# B&R Automation Studio project CombinedLinenSoiledA9KAN (part 10)

```iecst
			//###DK2012Jan12
			// Set statistic.
			IF _wPrevMsgStatisticSelect <> IFmnMsg.In.wMsgStatisticSelect THEN
				_wPrevMsgStatisticSelect := IFmnMsg.In.wMsgStatisticSelect;
				_xMsgStatisticSelectChanged := TRUE;
			END_IF;

			IF IFmnMsg.Trig.xRefreshStatistic OR _xRefreshStatistic THEN
				_msgStatisticNumShowIdx := _msgStatisticNumIdx;
				_msgStatisticTimeShowIdx := _msgStatisticTimeIdx;
				_wIFMsgStatisticCntNumShow := _wIFMsgStatisticCntNum;
				_wIFMsgStatisticCntTimeShow := _wIFMsgStatisticCntTime;
				IFmnMsg.Trig.xRefreshStatistic := FALSE;
				_xRefreshStatistic := FALSE;
				_xMsgStatisticSelectChanged := TRUE;
			END_IF;

			IF _xMsgStatisticSelectChanged THEN
				IF IFmnMsg.In.wMsgStatisticSelect = 0 THEN
					IFmnMsg.Out.wMsgStatisticCnt := _wIFMsgStatisticCntNumShow;
					FOR _wMsgListCnt := 0 TO MNMSG_MAX_IDX_VCMSGSTATLIST BY 1 DO
						_utfMsgTextTempFirst := UINT_TO_WSTRING(_msgStatisticNumShowIdx[_wMsgListCnt].wFunction_ID);
						_utfMsgTextTempSecond := ".";
						brwcsncat(ADR(_utfMsgTextTempFirst), ADR(_utfMsgTextTempSecond),
						UDINT_TO_UINT(brwcslen(ADR(_utfMsgTextTempSecond)) - (brwcslen(ADR(_utfMsgTextTempFirst)) + brwcslen(ADR(_utfMsgTextTempSecond)) - (SIZEOF(_utfMsgTextTempFirst) / 2 - 1))));
						_utfMsgTextTempSecond := UINT_TO_WSTRING(_msgStatisticNumShowIdx[_wMsgListCnt].wMsgNumber);
						brwcsncat(ADR(_utfMsgTextTempFirst), ADR(_utfMsgTextTempSecond),
						UDINT_TO_UINT(brwcslen(ADR(_utfMsgTextTempSecond)) - (brwcslen(ADR(_utfMsgTextTempFirst)) + brwcslen(ADR(_utfMsgTextTempSecond)) - (SIZEOF(_utfMsgTextTempFirst) / 2 - 1))));
						_utfMsgTextTempSecond := ".";
						brwcsncat(ADR(_utfMsgTextTempFirst), ADR(_utfMsgTextTempSecond),
						UDINT_TO_UINT(brwcslen(ADR(_utfMsgTextTempSecond)) - (brwcslen(ADR(_utfMsgTextTempFirst)) + brwcslen(ADR(_utfMsgTextTempSecond)) - (SIZEOF(_utfMsgTextTempFirst) / 2 - 1))));
						_utfMsgTextTempSecond := UINT_TO_WSTRING(_msgStatisticNumShowIdx[_wMsgListCnt].wInstance);
						brwcsncat(ADR(_utfMsgTextTempFirst), ADR(_utfMsgTextTempSecond),
						UDINT_TO_UINT(brwcslen(ADR(_utfMsgTextTempSecond)) - (brwcslen(ADR(_utfMsgTextTempFirst)) + brwcslen(ADR(_utfMsgTextTempSecond)) - (SIZEOF(_utfMsgTextTempFirst) / 2 - 1))));
						_utfMsgTextTempSecond := " ";
						brwcsncat(ADR(_utfMsgTextTempFirst), ADR(_utfMsgTextTempSecond),
						UDINT_TO_UINT(brwcslen(ADR(_utfMsgTextTempSecond)) - (brwcslen(ADR(_utfMsgTextTempFirst)) + brwcslen(ADR(_utfMsgTextTempSecond)) - (SIZEOF(_utfMsgTextTempFirst) / 2 - 1))));
						_wActFunctionID := _msgStatisticNumShowIdx[_wMsgListCnt].wFunction_ID;
						_wActMsgNumber := _msgStatisticNumShowIdx[_wMsgListCnt].wMsgNumber;
						_wActInstance := _msgStatisticNumShowIdx[_wMsgListCnt].wInstance;
						_actGetTxtFim;
						IF NOT((_wActFunctionID = 0) OR (_wActMsgNumber = 0)) THEN
							IFmnMsg.Out.MsgStatistic[_wMsgListCnt].utfMsgText := _utfMsgTextTempFirst;
							IFmnMsg.Out.MsgStatistic[_wMsgListCnt].lValue := _msgStatisticNumShowIdx[_wMsgListCnt].lValue;
						ELSE
							IFmnMsg.Out.MsgStatistic[_wMsgListCnt].utfMsgText := "";
							IFmnMsg.Out.MsgStatistic[_wMsgListCnt].lValue := 0;
						END_IF;
					END_FOR;
				END_IF;
				IF IFmnMsg.In.wMsgStatisticSelect = 1 THEN
					IFmnMsg.Out.wMsgStatisticCnt := _wIFMsgStatisticCntTimeShow;
					FOR _wMsgListCnt := 0 TO MNMSG_MAX_IDX_VCMSGSTATLIST BY 1 DO
						_utfMsgTextTempFirst := UINT_TO_WSTRING(_msgStatisticTimeShowIdx[_wMsgListCnt].wFunction_ID);
						_utfMsgTextTempSecond := ".";
						brwcsncat(ADR(_utfMsgTextTempFirst), ADR(_utfMsgTextTempSecond),
						UDINT_TO_UINT(brwcslen(ADR(_utfMsgTextTempSecond)) - (brwcslen(ADR(_utfMsgTextTempFirst)) + brwcslen(ADR(_utfMsgTextTempSecond)) - (SIZEOF(_utfMsgTextTempFirst) / 2 - 1))));
						_utfMsgTextTempSecond := UINT_TO_WSTRING(_msgStatisticTimeShowIdx[_wMsgListCnt].wMsgNumber);
						brwcsncat(ADR(_utfMsgTextTempFirst), ADR(_utfMsgTextTempSecond),
						UDINT_TO_UINT(brwcslen(ADR(_utfMsgTextTempSecond)) - (brwcslen(ADR(_utfMsgTextTempFirst)) + brwcslen(ADR(_utfMsgTextTempSecond)) - (SIZEOF(_utfMsgTextTempFirst) / 2 - 1))));
						_utfMsgTextTempSecond := ".";
						brwcsncat(ADR(_utfMsgTextTempFirst), ADR(_utfMsgTextTempSecond),
						UDINT_TO_UINT(brwcslen(ADR(_utfMsgTextTempSecond)) - (brwcslen(ADR(_utfMsgTextTempFirst)) + brwcslen(ADR(_utfMsgTextTempSecond)) - (SIZEOF(_utfMsgTextTempFirst) / 2 - 1))));
						_utfMsgTextTempSecond := UINT_TO_WSTRING(_msgStatisticTimeShowIdx[_wMsgListCnt].wInstance);
						brwcsncat(ADR(_utfMsgTextTempFirst), ADR(_utfMsgTextTempSecond),
						UDINT_TO_UINT(brwcslen(ADR(_utfMsgTextTempSecond)) - (brwcslen(ADR(_utfMsgTextTempFirst)) + brwcslen(ADR(_utfMsgTextTempSecond)) - (SIZEOF(_utfMsgTextTempFirst) / 2 - 1))));
						_utfMsgTextTempSecond := " ";
						brwcsncat(ADR(_utfMsgTextTempFirst), ADR(_utfMsgTextTempSecond),
						UDINT_TO_UINT(brwcslen(ADR(_utfMsgTextTempSecond)) - (brwcslen(ADR(_utfMsgTextTempFirst)) + brwcslen(ADR(_utfMsgTextTempSecond)) - (SIZEOF(_utfMsgTextTempFirst) / 2 - 1))));
						_wActFunctionID := _msgStatisticTimeShowIdx[_wMsgListCnt].wFunction_ID;
						_wActMsgNumber := _msgStatisticTimeShowIdx[_wMsgListCnt].wMsgNumber;
						_wActInstance := _msgStatisticTimeShowIdx[_wMsgListCnt].wInstance;
						_actGetTxtFim;
						IF NOT ((_wActFunctionID = 0) OR (_wActMsgNumber = 0)) THEN
							IFmnMsg.Out.MsgStatistic[_wMsgListCnt].utfMsgText := _utfMsgTextTempFirst;
							IFmnMsg.Out.MsgStatistic[_wMsgListCnt].lValue := _msgStatisticTimeShowIdx[_wMsgListCnt].lValue;
						ELSE
							IFmnMsg.Out.MsgStatistic[_wMsgListCnt].utfMsgText := "";
							IFmnMsg.Out.MsgStatistic[_wMsgListCnt].lValue := 0;
						END_IF;
					END_FOR;
				END_IF;
				_xMsgStatisticSelectChanged := FALSE;
			END_IF;
			//###DK2012Jan12

		END_IF

	ELSE	// _Plausibility.xOK

		// Horning for 500ms. After it has finished it will start again ten seconds later.
		_tonCrit1(IN := NOT _tonCrit2.Q, PT := T#500ms);
		_tonCrit2(IN := _tonCrit1.Q, PT := T#10s);

		IFmnMsg.Out.bHorn := SEL(NOT _tonCrit1.Q, 0, 1);	// Causes some horning now.

		IFmnMsg.Out.bLight := 1;

		// Meldung setzen

		IF _xNotOkFirstScan THEN

			_xNotOkFirstScan := FALSE;

			// Meldungsliste füllen

			brsmemset (ADR(mnMsgStatAd.Msg), 0, SIZEOF (mnMsgStatAd.Msg));

			_InsertMsgLine.AdrIntFaultList := ADR(mnMsgStatAd.Msg.MsgListFaultInt);
			_InsertMsgLine.AdrCntIntFault := ADR(mnMsgStatAd.Msg.MsgCntFaultInt);

			_dtHelp(enable := TRUE);

			_InsertMsgLine.Class := MNMSG_CLASS_INTFAULT;
			_InsertMsgLine.Insert := TRUE;
			_InsertMsgLine.MsgLine.bAckLevel := MNMSG_CLASS_NO_ACK;
			_InsertMsgLine.MsgLine.bInstance := 0;
			_InsertMsgLine.MsgLine.diAttr1 := 0;
			_InsertMsgLine.MsgLine.wFunction_ID := 2;
			_InsertMsgLine.MsgLine.wMsgNumber := MNMSG_MSG_SYSTEMFAULT;
			_InsertMsgLine.MsgLine.TimeStamp := _dtHelp.DT1;
			_InsertMsgLine();

			mnMsgStatAd.Msg.dtMsgIntFaultChanged := _dtHelp.DT1;

		END_IF

	END_IF;	// IFmnMsg.Out.xMnMsgReady

	////////////////////////////////////////////////////////////////////////////////////////////////////////////////////////////////////////////////////////////////////////////////////////////////////////////////////////////////////////////////////////////////////////////////////////////////////////////////////////////////////////////////////////////////////////////////////////////////////////////////////////////////////////////////////////////////////////////////////////////////////////////////////////////////////////////////////////////////////////////////////////////////////////////////////////////////////

	_LastExecute(enable := TRUE);
	_dtLastExecute := _LastExecute.DT1;

END_PROGRAM
```

#### _actGetTxtFim.st
```iecst
(********************************************************************
 * COPYRIGHT -- Herbert Kannegiesser GmbH
 ********************************************************************
 * Program: mnMsg
 * File: actGetTxtFim.st
 * Author: kuehne
 * Created: February 21, 2012
 ********************************************************************
 * Implementation of program mnMsg
 ********************************************************************)

(* Add a new action to your IEC program or library *)
ACTION _actGetTxtFim:
	IF _xMnTxtReady THEN
		_MsgTxtLine ACCESS IFmnTxt.Out.ptrFunctionTxtList;
		_BinSearchTxt.MsgTxtList := IFmnTxt.Out.ptrFunctionTxtList;
		_BinSearchTxt.wCntMsgTxt := IFmnTxt.Out.wCntFunctionTxt;
		_BinSearchTxt.wFunctionID := _wActFunctionID;
		_BinSearchTxt.wNumber := _wActMsgNumber;
		_BinSearchTxt.wInstance := _wActInstance;
		_BinSearchTxt.bTupel := 1;
		_BinSearchTxt();
		IF _BinSearchTxt.wStatus <> ERR_OK THEN
			brwcscat(ADR(_utfMsgTextTempFirst), ADR(""));
		ELSE
			_wTxtIdx := _BinSearchTxt.wMsgPos;
			_BinSearchCfg.wFunctionID := _wActFunctionID;
			_BinSearchCfg.wMsgNo := _wActMsgNumber;
			_BinSearchCfg.wInstance := _wActInstance;
			_BinSearchCfg();
			IF _BinSearchCfg.wStatus = ERR_OK THEN
				_wImageIdx := _BinSearchCfg.wMsgIdx;
				_utfMsgTextTempThird := "";
				_utfMsgTextTempThird := DINT_TO_WSTRING(_MsgImage[_wImageIdx].diMsgAttr1);
			ELSE
				_utfMsgTextTempThird := "{##AttrVar1}";
			END_IF;
			_utfMsgTextTempSecond := "";
			_fbMsgReplSubStr.utfStr := ADR(_MsgTxtLine[_wTxtIdx].utfText);
			_fbMsgReplSubStr.utfSubStr := ADR("{##AttrVar1}");
			_fbMsgReplSubStr.utfStrToReplWith := ADR(_utfMsgTextTempThird);
			_fbMsgReplSubStr.utfStrResult := ADR(_utfMsgTextTempSecond);
			_fbMsgReplSubStr();
			IF _BinSearchCfg.wStatus = ERR_OK THEN
				_wImageIdx := _BinSearchCfg.wMsgIdx;
				_utfMsgTextTempThird := "";
				_utfMsgTextTempThird := DINT_TO_WSTRING(_MsgImage[_wImageIdx].diMsgAttr2);
			ELSE
				_utfMsgTextTempThird := "{##AttrVar2}";
			END_IF;
			_utfMsgTextTempFourth := "";
			_utfMsgTextTempFourth := _utfMsgTextTempSecond;
			_utfMsgTextTempSecond := "";
			_fbMsgReplSubStr.utfStr := ADR(_utfMsgTextTempFourth);
			_fbMsgReplSubStr.utfSubStr := ADR("{##AttrVar2}");
			_fbMsgReplSubStr.utfStrToReplWith := ADR(_utfMsgTextTempThird);
			_fbMsgReplSubStr.utfStrResult := ADR(_utfMsgTextTempSecond);
			_fbMsgReplSubStr();
			IF _BinSearchCfg.wStatus = ERR_OK THEN
				_wImageIdx := _BinSearchCfg.wMsgIdx;
				_utfMsgTextTempThird := "";
				_utfMsgTextTempThird := STRING_TO_WSTRING(_MsgImage[_wImageIdx].sMsgAttrTxt);
			ELSE
				_utfMsgTextTempThird := "{##AttrTxt}";
			END_IF;
			_utfMsgTextTempFourth := "";
			_utfMsgTextTempFourth := _utfMsgTextTempSecond;
			_utfMsgTextTempSecond := "";
			_fbMsgReplSubStr.utfStr := ADR(_utfMsgTextTempFourth);
			_fbMsgReplSubStr.utfSubStr := ADR("{##AttrTxt}");
			_fbMsgReplSubStr.utfStrToReplWith := ADR(_utfMsgTextTempThird);
			_fbMsgReplSubStr.utfStrResult := ADR(_utfMsgTextTempSecond);
			_fbMsgReplSubStr();
			brwcsncat(ADR(_utfMsgTextTempFirst), ADR(_utfMsgTextTempSecond),
			UDINT_TO_UINT(brwcslen(ADR(_utfMsgTextTempSecond)) - (brwcslen(ADR(_utfMsgTextTempFirst)) + brwcslen(ADR(_utfMsgTextTempSecond)) - (SIZEOF(_utfMsgTextTempFirst) / 2 - 1))));
			_utfMsgTextTempSecond := "";
			_utfMsgTextTempSecond := " ";
			brwcsncat(ADR(_utfMsgTextTempFirst), ADR(_utfMsgTextTempSecond),
			UDINT_TO_UINT(brwcslen(ADR(_utfMsgTextTempSecond)) - (brwcslen(ADR(_utfMsgTextTempFirst)) + brwcslen(ADR(_utfMsgTextTempSecond)) - (SIZEOF(_utfMsgTextTempFirst) / 2 - 1))));
		END_IF;
		_MsgTxtLine ACCESS IFmnTxt.Out.ptrInstanceTxtList;
		_BinSearchTxt.MsgTxtList := IFmnTxt.Out.ptrInstanceTxtList;
		_BinSearchTxt.wCntMsgTxt := IFmnTxt.Out.wCntInstanceTxt;
		_BinSearchTxt.wFunctionID := _wActFunctionID;
		_BinSearchTxt.wNumber := _wActInstance;
		_BinSearchTxt.wInstance := 0;
		_BinSearchTxt.bTupel := 2;
		_BinSearchTxt();
		IF _BinSearchTxt.wStatus <> ERR_OK THEN
			brwcscat(ADR(_utfMsgTextTempFirst), ADR(""));
		ELSE
			_wTxtIdx := _BinSearchTxt.wMsgPos;
			_BinSearchCfg.wFunctionID := _wActFunctionID;
			_BinSearchCfg.wMsgNo := _wActMsgNumber;
			_BinSearchCfg.wInstance := _wActInstance;
			_BinSearchCfg();
			IF _BinSearchCfg.wStatus = ERR_OK THEN
				_wImageIdx := _BinSearchCfg.wMsgIdx;
				_utfMsgTextTempThird := "";
				_utfMsgTextTempThird := DINT_TO_WSTRING(_MsgImage[_wImageIdx].diMsgAttr1);
			ELSE
				_utfMsgTextTempThird := "{##AttrVar1}";
			END_IF;
			_utfMsgTextTempSecond := "";
			_fbMsgReplSubStr.utfStr := ADR(_MsgTxtLine[_wTxtIdx].utfText);
			_fbMsgReplSubStr.utfSubStr := ADR("{##AttrVar1}");
			_fbMsgReplSubStr.utfStrToReplWith := ADR(_utfMsgTextTempThird);
			_fbMsgReplSubStr.utfStrResult := ADR(_utfMsgTextTempSecond);
			_fbMsgReplSubStr();
			IF _BinSearchCfg.wStatus = ERR_OK THEN
				_wImageIdx := _BinSearchCfg.wMsgIdx;
				_utfMsgTextTempThird := "";
				_utfMsgTextTempThird := DINT_TO_WSTRING(_MsgImage[_wImageIdx].diMsgAttr2);
			ELSE
				_utfMsgTextTempThird := "{##AttrVar2}";
			END_IF;
			_utfMsgTextTempFourth := "";
			_utfMsgTextTempFourth := _utfMsgTextTempSecond;
			_utfMsgTextTempSecond := "";
			_fbMsgReplSubStr.utfStr := ADR(_utfMsgTextTempFourth);
			_fbMsgReplSubStr.utfSubStr := ADR("{##AttrVar2}");
			_fbMsgReplSubStr.utfStrToReplWith := ADR(_utfMsgTextTempThird);
			_fbMsgReplSubStr.utfStrResult := ADR(_utfMsgTextTempSecond);
			_fbMsgReplSubStr();
			IF _BinSearchCfg.wStatus = ERR_OK THEN
				_wImageIdx := _BinSearchCfg.wMsgIdx;
				_utfMsgTextTempThird := "";
				_utfMsgTextTempThird := STRING_TO_WSTRING(_MsgImage[_wImageIdx].sMsgAttrTxt);
			ELSE
				_utfMsgTextTempThird := "{##AttrTxt}";
			END_IF;
			_utfMsgTextTempFourth := "";
			_utfMsgTextTempFourth := _utfMsgTextTempSecond;
			_utfMsgTextTempSecond := "";
			_fbMsgReplSubStr.utfStr := ADR(_utfMsgTextTempFourth);
			_fbMsgReplSubStr.utfSubStr := ADR("{##AttrTxt}");
			_fbMsgReplSubStr.utfStrToReplWith := ADR(_utfMsgTextTempThird);
			_fbMsgReplSubStr.utfStrResult := ADR(_utfMsgTextTempSecond);
			_fbMsgReplSubStr();
			brwcsncat(ADR(_utfMsgTextTempFirst), ADR(_utfMsgTextTempSecond),
			UDINT_TO_UINT(brwcslen(ADR(_utfMsgTextTempSecond)) - (brwcslen(ADR(_utfMsgTextTempFirst)) + brwcslen(ADR(_utfMsgTextTempSecond)) - (SIZEOF(_utfMsgTextTempFirst) / 2 - 1))));
			_utfMsgTextTempSecond := "";
			_utfMsgTextTempSecond := " ";
			brwcsncat(ADR(_utfMsgTextTempFirst), ADR(_utfMsgTextTempSecond),
			UDINT_TO_UINT(brwcslen(ADR(_utfMsgTextTempSecond)) - (brwcslen(ADR(_utfMsgTextTempFirst)) + brwcslen(ADR(_utfMsgTextTempSecond)) - (SIZEOF(_utfMsgTextTempFirst) / 2 - 1))));
		END_IF;
		_MsgTxtLine ACCESS IFmnTxt.Out.ptrMessageTxtList;
		_BinSearchTxt.MsgTxtList := IFmnTxt.Out.ptrMessageTxtList;
		_BinSearchTxt.wCntMsgTxt := IFmnTxt.Out.wCntMessageTxt;
		_BinSearchTxt.wFunctionID := _wActFunctionID;
		_BinSearchTxt.wNumber := _wActMsgNumber;
		_BinSearchTxt.wInstance := _wActInstance;
		_BinSearchTxt.bTupel := 2;
		_BinSearchTxt();
		IF _BinSearchTxt.wStatus <> ERR_OK THEN
			brwcscat(ADR(_utfMsgTextTempFirst), ADR(""));
		ELSE
			_wTxtIdx := _BinSearchTxt.wMsgPos;
			_BinSearchCfg.wFunctionID := _wActFunctionID;
			_BinSearchCfg.wMsgNo := _wActMsgNumber;
			_BinSearchCfg.wInstance := _wActInstance;
			_BinSearchCfg();
			IF _BinSearchCfg.wStatus = ERR_OK THEN
				_wImageIdx := _BinSearchCfg.wMsgIdx;
				_utfMsgTextTempThird := "";
				_utfMsgTextTempThird := DINT_TO_WSTRING(_MsgImage[_wImageIdx].diMsgAttr1);
			ELSE
				_utfMsgTextTempThird := "{##AttrVar1}";
			END_IF;
			_utfMsgTextTempSecond := "";
			_fbMsgReplSubStr.utfStr := ADR(_MsgTxtLine[_wTxtIdx].utfText);
			_fbMsgReplSubStr.utfSubStr := ADR("{##AttrVar1}");
			_fbMsgReplSubStr.utfStrToReplWith := ADR(_utfMsgTextTempThird);
			_fbMsgReplSubStr.utfStrResult := ADR(_utfMsgTextTempSecond);
			_fbMsgReplSubStr();
			IF _BinSearchCfg.wStatus = ERR_OK THEN
				_wImageIdx := _BinSearchCfg.wMsgIdx;
				_utfMsgTextTempThird := "";
				_utfMsgTextTempThird := DINT_TO_WSTRING(_MsgImage[_wImageIdx].diMsgAttr2);
			ELSE
				_utfMsgTextTempThird := "{##AttrVar2}";
			END_IF;
			_utfMsgTextTempFourth := "";
			_utfMsgTextTempFourth := _utfMsgTextTempSecond;
			_utfMsgTextTempSecond := "";
			_fbMsgReplSubStr.utfStr := ADR(_utfMsgTextTempFourth);
			_fbMsgReplSubStr.utfSubStr := ADR("{##AttrVar2}");
			_fbMsgReplSubStr.utfStrToReplWith := ADR(_utfMsgTextTempThird);
			_fbMsgReplSubStr.utfStrResult := ADR(_utfMsgTextTempSecond);
			_fbMsgReplSubStr();
			IF _BinSearchCfg.wStatus = ERR_OK THEN
				_wImageIdx := _BinSearchCfg.wMsgIdx;
				_utfMsgTextTempThird := "";
				_utfMsgTextTempThird := STRING_TO_WSTRING(_MsgImage[_wImageIdx].sMsgAttrTxt);
			ELSE
				_utfMsgTextTempThird := "{##AttrTxt}";
			END_IF;
			_utfMsgTextTempFourth := "";
			_utfMsgTextTempFourth := _utfMsgTextTempSecond;
			_utfMsgTextTempSecond := "";
			_fbMsgReplSubStr.utfStr := ADR(_utfMsgTextTempFourth);
			_fbMsgReplSubStr.utfSubStr := ADR("{##AttrTxt}");
			_fbMsgReplSubStr.utfStrToReplWith := ADR(_utfMsgTextTempThird);
			_fbMsgReplSubStr.utfStrResult := ADR(_utfMsgTextTempSecond);
			_fbMsgReplSubStr();
			brwcsncat(ADR(_utfMsgTextTempFirst), ADR(_utfMsgTextTempSecond),
			UDINT_TO_UINT(brwcslen(ADR(_utfMsgTextTempSecond)) - (brwcslen(ADR(_utfMsgTextTempFirst)) + brwcslen(ADR(_utfMsgTextTempSecond)) - (SIZEOF(_utfMsgTextTempFirst) / 2 - 1))));
		END_IF;
	ELSE
		brwcscat(ADR(_utfMsgTextTempFirst), ADR(""));
	END_IF;
END_ACTION
```

#### _actGetTxtFimh.st
```iecst
(********************************************************************
 * COPYRIGHT -- Herbert Kannegiesser GmbH
 ********************************************************************
 * Program: mnMsg
 * File: actGetTxtFimh.st
 * Author: kuehne
 * Created: February 22, 2012
 ********************************************************************
 * Implementation of program mnMsg
 ********************************************************************)

 (* Add a new action to your IEC program or library *)
ACTION _actGetTxtFimh:
	IF _xMnTxtReady THEN
		_MsgTxtLine ACCESS IFmnTxt.Out.ptrFunctionTxtList;
		_BinSearchTxt.MsgTxtList := IFmnTxt.Out.ptrFunctionTxtList;
		_BinSearchTxt.wCntMsgTxt := IFmnTxt.Out.wCntFunctionTxt;
		_BinSearchTxt.wFunctionID := _wActFunctionID;
		_BinSearchTxt.wNumber := _wActMsgNumber;
		_BinSearchTxt.wInstance := _wActInstance;
		_BinSearchTxt.bTupel := 1;
		_BinSearchTxt();
		IF _BinSearchTxt.wStatus <> ERR_OK THEN
			brwcscat(ADR(_utfMsgTextTempFirst), ADR(""));
		ELSE
			_wTxtIdx := _BinSearchTxt.wMsgPos;
			_utfMsgTextTempSecond := "";
			_utfMsgTextTempThird := "";
			_utfMsgTextTempThird := DINT_TO_WSTRING(_diActAttr1);
			_fbMsgReplSubStr.utfStr := ADR(_MsgTxtLine[_wTxtIdx].utfText);
			_fbMsgReplSubStr.utfSubStr := ADR("{##AttrVar1}");
			_fbMsgReplSubStr.utfStrToReplWith := ADR(_utfMsgTextTempThird);
			_fbMsgReplSubStr.utfStrResult := ADR(_utfMsgTextTempSecond);
			_fbMsgReplSubStr();
			_utfMsgTextTempThird := "";
			_utfMsgTextTempFourth := "";
			_utfMsgTextTempFourth := _utfMsgTextTempSecond;
			_utfMsgTextTempSecond := "";
			_utfMsgTextTempThird := DINT_TO_WSTRING(_diActAttr2);
			_fbMsgReplSubStr.utfStr := ADR(_utfMsgTextTempFourth);
			_fbMsgReplSubStr.utfSubStr := ADR("{##AttrVar2}");
			_fbMsgReplSubStr.utfStrToReplWith := ADR(_utfMsgTextTempThird);
			_fbMsgReplSubStr.utfStrResult := ADR(_utfMsgTextTempSecond);
			_fbMsgReplSubStr();
			_utfMsgTextTempThird := "";
			_utfMsgTextTempFourth := "";
			_utfMsgTextTempFourth := _utfMsgTextTempSecond;
			_utfMsgTextTempSecond := "";
			_utfMsgTextTempThird := STRING_TO_WSTRING(_sActAttrTxt);
			_fbMsgReplSubStr.utfStr := ADR(_utfMsgTextTempFourth);
			_fbMsgReplSubStr.utfSubStr := ADR("{##AttrTxt}");
			_fbMsgReplSubStr.utfStrToReplWith := ADR(_utfMsgTextTempThird);
			_fbMsgReplSubStr.utfStrResult := ADR(_utfMsgTextTempSecond);
			_fbMsgReplSubStr();
			brwcsncat(ADR(_utfMsgTextTempFirst), ADR(_utfMsgTextTempSecond),
			UDINT_TO_UINT(brwcslen(ADR(_utfMsgTextTempSecond)) - (brwcslen(ADR(_utfMsgTextTempFirst)) + brwcslen(ADR(_utfMsgTextTempSecond)) - (SIZEOF(_utfMsgTextTempFirst) / 2 - 1))));
			_utfMsgTextTempSecond := "";
			_utfMsgTextTempSecond := " ";
			brwcsncat(ADR(_utfMsgTextTempFirst), ADR(_utfMsgTextTempSecond),
			UDINT_TO_UINT(brwcslen(ADR(_utfMsgTextTempSecond)) - (brwcslen(ADR(_utfMsgTextTempFirst)) + brwcslen(ADR(_utfMsgTextTempSecond)) - (SIZEOF(_utfMsgTextTempFirst) / 2 - 1))));
		END_IF;
		_MsgTxtLine ACCESS IFmnTxt.Out.ptrInstanceTxtList;
		_BinSearchTxt.MsgTxtList := IFmnTxt.Out.ptrInstanceTxtList;
		_BinSearchTxt.wCntMsgTxt := IFmnTxt.Out.wCntInstanceTxt;
		_BinSearchTxt.wFunctionID := _wActFunctionID;
		_BinSearchTxt.wNumber := _wActInstance;
		_BinSearchTxt.wInstance := 0;
		_BinSearchTxt.bTupel := 2;
		_BinSearchTxt();
		IF _BinSearchTxt.wStatus <> ERR_OK THEN
			brwcscat(ADR(_utfMsgTextTempFirst), ADR(""));
		ELSE
			_wTxtIdx := _BinSearchTxt.wMsgPos;
			_utfMsgTextTempSecond := "";
			_utfMsgTextTempThird := "";
			_utfMsgTextTempThird := DINT_TO_WSTRING(_diActAttr1);
			_fbMsgReplSubStr.utfStr := ADR(_MsgTxtLine[_wTxtIdx].utfText);
			_fbMsgReplSubStr.utfSubStr := ADR("{##AttrVar1}");
			_fbMsgReplSubStr.utfStrToReplWith := ADR(_utfMsgTextTempThird);
			_fbMsgReplSubStr.utfStrResult := ADR(_utfMsgTextTempSecond);
			_fbMsgReplSubStr();
			_utfMsgTextTempThird := "";
			_utfMsgTextTempFourth := "";
			_utfMsgTextTempFourth := _utfMsgTextTempSecond;
			_utfMsgTextTempSecond := "";
			_utfMsgTextTempThird := DINT_TO_WSTRING(_diActAttr2);
			_fbMsgReplSubStr.utfStr := ADR(_utfMsgTextTempFourth);
			_fbMsgReplSubStr.utfSubStr := ADR("{##AttrVar2}");
			_fbMsgReplSubStr.utfStrToReplWith := ADR(_utfMsgTextTempThird);
			_fbMsgReplSubStr.utfStrResult := ADR(_utfMsgTextTempSecond);
			_fbMsgReplSubStr();
			_utfMsgTextTempThird := "";
			_utfMsgTextTempFourth := "";
			_utfMsgTextTempFourth := _utfMsgTextTempSecond;
			_utfMsgTextTempSecond := "";
			_utfMsgTextTempThird := STRING_TO_WSTRING(_sActAttrTxt);
			_fbMsgReplSubStr.utfStr := ADR(_utfMsgTextTempFourth);
			_fbMsgReplSubStr.utfSubStr := ADR("{##AttrTxt}");
			_fbMsgReplSubStr.utfStrToReplWith := ADR(_utfMsgTextTempThird);
			_fbMsgReplSubStr.utfStrResult := ADR(_utfMsgTextTempSecond);
			_fbMsgReplSubStr();
			brwcsncat(ADR(_utfMsgTextTempFirst), ADR(_utfMsgTextTempSecond),
			UDINT_TO_UINT(brwcslen(ADR(_utfMsgTextTempSecond)) - (brwcslen(ADR(_utfMsgTextTempFirst)) + brwcslen(ADR(_utfMsgTextTempSecond)) - (SIZEOF(_utfMsgTextTempFirst) / 2 - 1))));
			_utfMsgTextTempSecond := "";
			_utfMsgTextTempSecond := " ";
			brwcsncat(ADR(_utfMsgTextTempFirst), ADR(_utfMsgTextTempSecond),
			UDINT_TO_UINT(brwcslen(ADR(_utfMsgTextTempSecond)) - (brwcslen(ADR(_utfMsgTextTempFirst)) + brwcslen(ADR(_utfMsgTextTempSecond)) - (SIZEOF(_utfMsgTextTempFirst) / 2 - 1))));
		END_IF;
		_MsgTxtLine ACCESS IFmnTxt.Out.ptrMessageTxtList;
		_BinSearchTxt.MsgTxtList := IFmnTxt.Out.ptrMessageTxtList;
		_BinSearchTxt.wCntMsgTxt := IFmnTxt.Out.wCntMessageTxt;
		_BinSearchTxt.wFunctionID := _wActFunctionID;
		_BinSearchTxt.wNumber := _wActMsgNumber;
		_BinSearchTxt.wInstance := _wActInstance;
		_BinSearchTxt.bTupel := 2;
		_BinSearchTxt();
		IF _BinSearchTxt.wStatus <> ERR_OK THEN
			brwcscat(ADR(_utfMsgTextTempFirst), ADR(""));
		ELSE
			_wTxtIdx := _BinSearchTxt.wMsgPos;
			_utfMsgTextTempSecond := "";
			_utfMsgTextTempThird := "";
			_utfMsgTextTempThird := DINT_TO_WSTRING(_diActAttr1);
			_fbMsgReplSubStr.utfStr := ADR(_MsgTxtLine[_wTxtIdx].utfText);
			_fbMsgReplSubStr.utfSubStr := ADR("{##AttrVar1}");
			_fbMsgReplSubStr.utfStrToReplWith := ADR(_utfMsgTextTempThird);
			_fbMsgReplSubStr.utfStrResult := ADR(_utfMsgTextTempSecond);
			_fbMsgReplSubStr();
			_utfMsgTextTempThird := "";
			_utfMsgTextTempFourth := "";
			_utfMsgTextTempFourth := _utfMsgTextTempSecond;
			_utfMsgTextTempSecond := "";
			_utfMsgTextTempThird := DINT_TO_WSTRING(_diActAttr2);
			_fbMsgReplSubStr.utfStr := ADR(_utfMsgTextTempFourth);
			_fbMsgReplSubStr.utfSubStr := ADR("{##AttrVar2}");
			_fbMsgReplSubStr.utfStrToReplWith := ADR(_utfMsgTextTempThird);
			_fbMsgReplSubStr.utfStrResult := ADR(_utfMsgTextTempSecond);
			_fbMsgReplSubStr();
			_utfMsgTextTempThird := "";
			_utfMsgTextTempFourth := "";
			_utfMsgTextTempFourth := _utfMsgTextTempSecond;
			_utfMsgTextTempSecond := "";
			_utfMsgTextTempThird := STRING_TO_WSTRING(_sActAttrTxt);
			_fbMsgReplSubStr.utfStr := ADR(_utfMsgTextTempFourth);
			_fbMsgReplSubStr.utfSubStr := ADR("{##AttrTxt}");
			_fbMsgReplSubStr.utfStrToReplWith := ADR(_utfMsgTextTempThird);
			_fbMsgReplSubStr.utfStrResult := ADR(_utfMsgTextTempSecond);
			_fbMsgReplSubStr();
			brwcsncat(ADR(_utfMsgTextTempFirst), ADR(_utfMsgTextTempSecond),
			UDINT_TO_UINT(brwcslen(ADR(_utfMsgTextTempSecond)) - (brwcslen(ADR(_utfMsgTextTempFirst)) + brwcslen(ADR(_utfMsgTextTempSecond)) - (SIZEOF(_utfMsgTextTempFirst) / 2 - 1))));
		END_IF;
		// wcscat(ADR(_utfMsgTextTempFirst), ADR("internal error"));	//Also for test
		_MsgHelpTxtLine ACCESS IFmnTxt.Out.ptrMessageHelpTxtList;
		_BinSearchHelpTxt.MsgHelpTxtList := IFmnTxt.Out.ptrMessageHelpTxtList;
		_BinSearchHelpTxt.wCntMsgHelpTxt := IFmnTxt.Out.wCntMessageHlpTxt;
		_BinSearchHelpTxt.wFunctionID := _wActFunctionID;
		_BinSearchHelpTxt.wNumber := _wActMsgNumber;
		_BinSearchHelpTxt.wInstance := _wActInstance;
		_BinSearchHelpTxt.bTupel := 2;
		_BinSearchHelpTxt();
		IF _BinSearchHelpTxt.wStatus <> ERR_OK THEN
			_utfMsgTextTempSecond := "";
		ELSE
			_wTxtIdx := _BinSearchHelpTxt.wMsgPos;
			_utfMsgTextTempSecond := "";
			_utfMsgTextTempThird := "";
			_utfMsgTextTempThird := DINT_TO_WSTRING(_diActAttr1);
			_fbMsgReplSubStr.utfStr := ADR(_MsgHelpTxtLine[_wTxtIdx].utfText);
			_fbMsgReplSubStr.utfSubStr := ADR("{##AttrVar1}");
			_fbMsgReplSubStr.utfStrToReplWith := ADR(_utfMsgTextTempThird);
			_fbMsgReplSubStr.utfStrResult := ADR(_utfMsgTextTempSecond);
			_fbMsgReplSubStr();
			_utfMsgTextTempThird := "";
			_utfMsgTextTempFourth := "";
			_utfMsgTextTempFourth := _utfMsgTextTempSecond;
			_utfMsgTextTempSecond := "";
			_utfMsgTextTempThird := DINT_TO_WSTRING(_diActAttr2);
			_fbMsgReplSubStr.utfStr := ADR(_utfMsgTextTempFourth);
			_fbMsgReplSubStr.utfSubStr := ADR("{##AttrVar2}");
			_fbMsgReplSubStr.utfStrToReplWith := ADR(_utfMsgTextTempThird);
			_fbMsgReplSubStr.utfStrResult := ADR(_utfMsgTextTempSecond);
			_fbMsgReplSubStr();
			_utfMsgTextTempThird := "";
			_utfMsgTextTempFourth := "";
			_utfMsgTextTempFourth := _utfMsgTextTempSecond;
			_utfMsgTextTempSecond := "";
			_utfMsgTextTempThird := STRING_TO_WSTRING(_sActAttrTxt);
			_fbMsgReplSubStr.utfStr := ADR(_utfMsgTextTempFourth);
			_fbMsgReplSubStr.utfSubStr := ADR("{##AttrTxt}");
			_fbMsgReplSubStr.utfStrToReplWith := ADR(_utfMsgTextTempThird);
			_fbMsgReplSubStr.utfStrResult := ADR(_utfMsgTextTempSecond);
			_fbMsgReplSubStr();
		END_IF;
	ELSE
		brwcscat(ADR(_utfMsgTextTempFirst), ADR(""));
		brwcscat(ADR(_utfMsgTextTempSecond), ADR(""));
	END_IF; // IF _xMnTxtReady THEN
END_ACTION
```

- Library Logical/Mewa/KGFramework/Pkg_mnMsg/KGlibMsg (IEC) - A new source library (no source held here)

### mnMsg-History.txt
```
1.00.0	01.07.2011	Neu
1.01.0	02.07.2011	Index für kgMsgStatus ist wählbar
1.02.0	29.07.2011	Setzten des Machinestate.xFault
1.02.1	23.08.2011	Einzelquittierung Low-und High-Word getauscht
			Hupen-Ansteuerung Faktor 1000 für Zeitbasis ergänzt

1.03.0	08.09.2011	- Mit der Compilerdirektive "-D Test" können Testmeldungen
			  erzeugt werden.
			- Fehler behoben. Es wurde kein Änderungs-Event erzeugt, wenn eine Meldungsklasse > 0 ist
			- MNMSG_IDX_KGMSGSTATTEST eingeführt, um Testmeldungen erzeugen zu können.

1.04.0	20.09.2011	- Schaut jetzt auf mnParamStatAd.xParamOK, setzt Version 0.5 von mnParam voraus
1.05.0	20.10.2011  - Umstellung auf AS 3.0.90. Entfernung der InOut-Elemente im Interface
1.06.0	20.12.2011	- Ringbuffer aus KGstandard verwenden
1.07.1	22.12.2011	- Fehler im Init-Up (Pointer für Ringbuffer) behoben
1.07.2	19.01.2012	- Seitenumschaltung für MsgHistList
1.07.3	25.01.2012	- In MsgList werden Attribute eingefügt
1.07.4	27.01.2012	- Attribute werden in alle Text-Listen eingefügt, neue bEvent Vergabe in HistList
1.07.5	17.02.2012	- RB aus KGstdLib für HistList, noch Ungenauigkeiten bei Überlauf
1.08.1	29.02.2012	- Cleaned-up code, RB can be read properly
1.09.0	01.03.2012	- Kommandokanal zum PC an den neuen Standard angepasst
					- Überflüssige Ringbuffer entfernt
					- Test entfernt
		02.03.2012	- Schnittstellen gekapselt.
					- Kommandos an IFmnMsg bereinigt. Auch für die Visu.
					- Der Test-Teil ist wieder entfallen, da das Framework einen Testadapter erhält.
1.10.0	03.03.2012	- MNMSG_RUN_VC eingeführt. Damit ist die Aufbereitung der VC-Listen abschaltbar.
					- Die Meldungsstatistik wird auf die Version der Konfiguration hin überwacht.
1.11.0	06.03.2012	- Bugfix
					- Kompatibel mit mnTest
1.11.1	07.03.2012	- Bugfix Wartungsmeldungen. Wurden nicht eingetragen
					- Hupe wird als Status ausgegeben
1.11.3	20.03.2012	- Version von Dirk Kühne
1.11.4	20.03.2012	- Gemerget
1.11.5	20.03.2012	- Bugfix Statistik löschen
					- Abhängigkeiten ergänzt
1.11.6	20.03.2012	- asBRWStr statt asWStr
1.11.7	23.03.2012	- Bugfix. Wartungsmeldung hat geflattert.
1.11.8	23.03.2012	- Zeitstempel für geänderte Meldungslisten feiner aufgelöst.
```

### CfgMsgStat.mnMsg.txt
```
;****************************
; Meldungsmanager mnMsg
;*****************************
00002, 01000, 00000, 00000;
00002, 01003, 00000, 00000;
```

### Package Logical/Mewa/KGFramework/Pkg_mnParam - Parameter-Manager

### mnParam.typ - Package data types
```iecst
(********************************************************************
 * COPYRIGHT -- Microsoft
 ********************************************************************
 * Package: Pkg_mnParam_Test
 * File: mnParam.typ
 * Author: hunholz
 * Created: July 23, 2011
 ********************************************************************
 * Data types of package Pkg_mnParam_Test
 ********************************************************************)

TYPE
	mnParamStatAd_typ : 	STRUCT
		xParamOK : BOOL;
		dtExportContent : DATE_AND_TIME;
		HeaderVersion : mnParam_HeaderVersionRow_typ;
		utfMachineNumber : WSTRING[15];
		utfMachineName : WSTRING[31];
		sPkgVersion : STRING[10];
		wCntFilesImportOK : UINT;
		wCntFilesImportFailed : UINT;
		wCntFilesImportFound : UINT;
	END_STRUCT;
END_TYPE

(*INTERFACE*)

TYPE
	mnParam_EditNumValue_typ : 	STRUCT
		rVal : ARRAY[1..MNPARAM_CNT_EDITROWS]OF REAL;
		xSave : ARRAY[1..MNPARAM_CNT_EDITROWS]OF BOOL;
		wIdx : ARRAY[1..MNPARAM_CNT_EDITROWS]OF UINT;
	END_STRUCT;
	mnParam_EditStrValue_typ : 	STRUCT
		utfVal : ARRAY[1..MNPARAM_CNT_EDITROWS]OF WSTRING[31];
		xSave : ARRAY[1..MNPARAM_CNT_EDITROWS]OF BOOL;
		wIdx : ARRAY[1..MNPARAM_CNT_EDITROWS]OF UINT;
	END_STRUCT;
	IFmnParamOutEditNumAttr_typ : 	STRUCT
		wType : UINT;
		wParIdx : UINT;
		wFunctionID : UINT;
		wParamNo : UINT;
		wArrIdx : ARRAY[1..4]OF UINT;
		bWriteAccess : USINT;
		bReadAccess : USINT;
		wUnit : UINT;
		utfParameterName : WSTRING[63];
		utfParameterHelpTxt : WSTRING[255];
		sUnit : STRING[11];
		rMin : REAL;
		rMax : REAL;
		rDefault : REAL;
		lDigits : UDINT;
	END_STRUCT;
	IFmnParamOutEditStrAttr_typ : 	STRUCT
		wType : UINT;
		wParIdx : UINT;
		wFunctionID : UINT;
		wParamNo : UINT;
		wArrIdx : ARRAY[1..4]OF UINT;
		bWriteAccess : USINT;
		bReadAccess : USINT;
		utfParameterName : WSTRING[63];
		utfParameterHelpTxt : WSTRING[255];
		utfDefault : WSTRING[31];
		wMaxLength : UINT;
	END_STRUCT;
	IFmnParamOutEdit_typ : 	STRUCT
		wStatus : UINT;
		bContainer : USINT;
		bCntNumRows : USINT;
		bCntStrRows : USINT;
		bReserve : USINT;
		wContainerInstance : UINT;
		wRowStrOffset : UINT;
		wRowNumOffset : UINT;
		lPtrEditNumValues : UDINT;
		lPtrEditStrValues : UDINT;
		AttrNum : ARRAY[1..MNPARAM_CNT_EDITROWS]OF IFmnParamOutEditNumAttr_typ;
		AttrStr : ARRAY[1..MNPARAM_CNT_EDITROWS]OF IFmnParamOutEditStrAttr_typ;
		wCntFilesImportOK : UINT;
		wCntFilesImportFailed : UINT;
		wCntFilesImportFound : UINT;
		wCntNamelist : UINT;
		wIdxContainerNamelist : UINT;
		wParIdxNamelist : UINT;
		wNameListNo : ARRAY[1..MNPARAM_CNT_NAMELIST]OF UINT;
		utfNameListName : ARRAY[1..MNPARAM_CNT_NAMELIST]OF WSTRING[39];
	END_STRUCT;
	IFmnParamOut_typ : 	STRUCT
		utfMachineNumber : WSTRING[15];
		xParamOK : BOOL;
		HeaderVersion : mnParam_HeaderVersionRow_typ;
		Edit : IFmnParamOutEdit_typ;
	END_STRUCT;
	IFmnParamInEdit_typ : 	STRUCT
		wCommand : UINT;
		bContainer : USINT;
		bCntNumRows : USINT;
		bCntStrRows : USINT;
		bLocUnit : USINT;
		bUserLevel : USINT;
		bSelectModeNum : USINT;
		bSelectModeStr : USINT;
		wContainerInstance : UINT;
		wContainerInstanceFrom : UINT;
		wRowStrOffset : UINT;
		wRowNumOffset : UINT;
		wSelParIdxNum : ARRAY[1..MNPARAM_CNT_EDITROWS]OF UINT;
		wSelParArrIdxNum : ARRAY[1..MNPARAM_CNT_EDITROWS,1..4]OF UINT;
		wSelParIdxStr : ARRAY[1..MNPARAM_CNT_EDITROWS]OF UINT;
		wSelParArrIdxStr : ARRAY[1..MNPARAM_CNT_EDITROWS,1..4]OF UINT;
		wSelIdxContainerNamelist : UINT;
		wSelParIdxNamelist : UINT;
	END_STRUCT;
	IFmnParamIn_typ : 	STRUCT
		Edit : IFmnParamInEdit_typ;
	END_STRUCT;
	IFmnParam_typ : 	STRUCT
		In : IFmnParamIn_typ;
		Out : IFmnParamOut_typ;
	END_STRUCT;
END_TYPE
```

### mnParam.var - Package variables
```iecst
(********************************************************************
 * COPYRIGHT -- Microsoft
 ********************************************************************
 * Package: PkgMNPARAM_Test
 * File: mnParam.var
 * Author: hunholz
 * Created: July 23, 2011
 ********************************************************************
 * Variables of package PkgMNPARAM_Test
 ********************************************************************)
(*Konstanten*)
VAR CONSTANT
	MNPARAM_FUNCTIONID : UINT := 1; (*Entsprechend Zuordnungsliste*)
	MNPARAM_PATH_PM : STRING[15] := 'PM\';
	MNPARAM_PATH_EXPORT : STRING[15] := 'PM\Export\';
	MNPARAM_PATH_IMPORT : STRING[15] := 'PM\Import\';
	MNPARAM_FILESUFF : STRING[7] := '.csv';
END_VAR
(*Kommandos*)
VAR CONSTANT
	MNPARAM_CMD_NOCOMMAND : UINT := 0;
	MNPARAM_CMD_IMPORT : UINT := 1;
	MNPARAM_CMD_DELETE : UINT := 2;
	MNPARAM_CMD_FILLEDITOR : UINT := 3;
	MNPARAM_CMD_SAVEEDITOR : UINT := 4;
	MNPARAM_CMD_CREATE_INDCONT : UINT := 5;
	MNPARAM_CMD_DELETE_INDCONT : UINT := 6;
	MNPARAM_CMD_COPY_INDCONT : UINT := 7;
	MNPARAM_CMD_BACKUP : UINT := 8;
	MNPARAM_CMD_RESTORE : UINT := 9;
	MNPARAM_CMD_FILLNAMELIST : UINT := 10;
	MNPARAM_CMD_MAX : UINT := 59999;
	MNPARAM_STAT_NOCOMMAND : UINT := 0;
	MNPARAM_STAT_FILLEDITOR_OK : UINT := 3;
	MNPARAM_STAT_SAVEEDITOR_OK : UINT := 4;
	MNPARAM_STAT_CREATE_INDCONT_OK : UINT := 5;
	MNPARAM_STAT_DELETE_INDCONT_OK : UINT := 6;
	MNPARAM_STAT_COPY_INDCONT_OK : UINT := 7;
	MNPARAM_STAT_BACKUP_OK : UINT := 8;
	MNPARAM_STAT_RESTORE_OK : UINT := 9;
	MNPARAM_STAT_FILLNAMELIST_OK : UINT := 10;
	MNPARAM_STAT_DIREMPTY : UINT := 60000;
	MNPARAM_STAT_WRONGIDX : UINT := 60001;
	MNPARAM_STAT_DELPARFAULT : UINT := 60002;
	MNPARAM_STAT_DELDEFFAULT : UINT := 60003;
	MNPARAM_STAT_NUMPARNOTFOUND : UINT := 60004;
	MNPARAM_STAT_WRITEPROTECTED : UINT := 60005;
	MNPARAM_STAT_STRPARNOTFOUND : UINT := 60006;
	MNPARAM_STAT_BINPARNOTFOUN : UINT := 60007;
	MNPARAM_STAT_DELNUMPAR : UINT := 60008;
	MNPARAM_STAT_DELSTRPAR : UINT := 60009;
	MNPARAM_STAT_DELBINPAR : UINT := 60010;
	MNPARAM_STAT_DELFILE : UINT := 60011;
	MNPARAM_STAT_IMPDIRREAD : UINT := 60020;
	MNPARAM_STAT_IMPFILENOTFND : UINT := 60021;
	MNPARAM_STAT_IMPALLOCMEM : UINT := 60022;
	MNPARAM_STAT_IMPOPENFILE : UINT := 60023;
	MNPARAM_STAT_IMPREADFILE : UINT := 60024;
	MNPARAM_STAT_IMPCNTLINES : UINT := 60025;
	MNPARAM_STAT_IMPTYPE : UINT := 60026;
	MNPARAM_STAT_IMPMACHINENO : UINT := 60027;
	MNPARAM_STAT_IMPROOT : UINT := 60028;
	MNPARAM_STAT_SYSERROR : UINT := 60029;
	MNPARAM_STAT_IMPALLOCMEMN : UINT := 60030;
	MNPARAM_STAT_IMPALLOCMEMS : UINT := 60031;
	MNPARAM_STAT_IMPREADNUM : UINT := 60032;
	MNPARAM_STAT_IMPREADSTR : UINT := 60033;
	MNPARAM_STAT_IMPREADBIN : UINT := 60034;
	MNPARAM_STAT_IMPWRITENUM : UINT := 60035;
	MNPARAM_STAT_IMPWRITESTR : UINT := 60036;
	MNPARAM_STAT_IMPWRITEBIN : UINT := 60037;
	MNPARAM_STAT_EXPALLOCMEMCSV : UINT := 60038;
	MNPARAM_STAT_CREATECSV : UINT := 60039;
	MNPARAM_STAT_OPENCSV : UINT := 60040;
	MNPARAM_STAT_WRITECSV : UINT := 60041;
	MNPARAM_STAT_CLOSECSV : UINT := 60042;
	MNPARAM_STAT_NULLPOINTER : UINT := 60043; (*Nullpointerfehler*)
	MNPARAM_STAT_EXPFREEMEM : UINT := 60044; (*Speicher für Exportdatei konnte nicht wieder frei gegeben werden*)
	MNPARAM_STAT_CONTAINER_NOT_VALID : UINT := 60045; (*Container ID ist nicht gültig*)
	MNPARAM_STAT_CONTINST_NOT_VALID : UINT := 60046; (*Containerinstanz ist nich gültig*)
	MNPARAM_STAT_CONTINST_NOT_EXIST : UINT := 60047; (*Containerinstanz existiert nicht*)
	MNPARAM_STAT_CONTINST_EMPTY : UINT := 60048; (*Container ist leer*)
	MNPARAM_STAT_FREEMEM : UINT := 60049;
	MNPARAM_STAT_DIRREAD : UINT := 60050;
	MNPARAM_STAT_NOUSBSTICK : UINT := 60051;
	MNPARAM_STAT_NOIMPORTDIR : UINT := 60052;
	MNPARAM_STAT_LINKUSB : UINT := 60053;
	MNPARAM_STAT_CREATEDIR : UINT := 60054;
	MNPARAM_STAT_COPY : UINT := 60055;
	MNPARAM_STAT_CONTINST_EXIST : UINT := 60056; (*Containerinstanz existiert bereits*)
	MNPARAM_STAT_FILENOTSUPPORTED : UINT := 60057; (*Datei kann nicht importiert werden*)
	MNPARAM_STAT_NOVERSION : UINT := 60058; (*Keine Version in der Datei*)
END_VAR
(*Meldungen*)
VAR CONSTANT
	MNPARAM_MSG_WARN_DELETE : UINT := 2;
	MNPARAM_MSG_WARN_IMPORT : UINT := 1;
	MNPARAM_MSG_WARN_FILLEDITOR : UINT := 3;
	MNPARAM_MSG_WARN_SAVEEDITOR : UINT := 4;
	MNPARAM_MSG_WARN_BACKUP : UINT := 5;
	MNPARAM_MSG_WARN_CREATE : UINT := 6;
	MNPARAM_MSG_WARN_COPY : UINT := 7;
	MNPARAM_MSG_WARN_IMPORTFAILED : UINT := 9;
	MNPARAM_MSG_SYSTEMERROR : UINT := 20000;
END_VAR
(*Auswahlmodi für Parameter*)
VAR CONSTANT
	MNPARAM_SELECTMODE_LINEAR : USINT := 0;
	MNPARAM_SELECTMODE_BYIDX : USINT := 1;
END_VAR
(*Importmodi*)
VAR CONSTANT
	MNPARAM_IMPORT_DIFFERENCE : UDINT := 0; (*Es werden nur die Daten verändert, die in der Importdatei stehen.*)
	MNPARAM_IMPORT_RESTORE : UDINT := 1; (*Vor dem Import der Daten, werden alle Daten des Containers auf Default zurückgesetzt.*)
END_VAR
(*Modi zum Prüfen der Maschinennummer im Datencontainer*)
VAR CONSTANT
	MNPARAM_CMNO_CHECK : UINT := 0; (*Datencontainer mit falscher Maschinennummer werden nicht importiert.*)
	MNPARAM_CMNO_CHECKNOT : UINT := 1; (*Datencontainer werden ohne Prüfung der Maschinennummer importiert.*)
END_VAR
(*Ungueltige Maschinennummer*)
VAR CONSTANT
	MNPARAM_INVALID_MACHINENO : WSTRING[15] := "dummy";
END_VAR
(*Interface-Variablen*)
VAR
	IFmnParam : IFmnParam_typ;
	mnParamCmd : KG_Cmd_typ;
	mnParamStat : Stat_typ;
	mnParamStatAd : mnParamStatAd_typ;
END_VAR
```

### Program Logical/Mewa/KGFramework/Pkg_mnParam/mnParam (IEC) - Parameter Manager
